{attribute 'GeneratedUsingTerminal: AX8206-0100-0101-0101'}
{attribute addProperty BoxType "AX8206-0100-0101-0101"}
{attribute addProperty Id "Ch_B_ControlwordAT %Q*UINT2"}
{attribute addProperty CRC "1382696952"}
{attribute addProperty Size "2"}
TYPE Ch_B_AxisMain_Outputs_526A47F8 :
STRUCT
	{attribute addProperty Name "Ch_B_Controlword"}
	Ch_B_Controlword AT %Q* : UINT;
END_STRUCT
END_TYPE

(* stored: Version 1.2.0.0, ProductVersion 3.1.4024.9
   DUT Ch_B_AxisMain_Outputs_526A47F8: Id {21910390-d76b-4534-8916-a9e1a79e65ce} *)
